{attribute 'pack_mode' := '1'}
TYPE DisableAllAxes EXTENDS IncomingMessage :
STRUCT
END_STRUCT
END_TYPE

(* stored: Version 1.1.0.1, ProductVersion 3.1.4022.12
   DUT DisableAllAxes: Id {45c8f6d1-a375-4c15-af2b-d88e45e54997} *)
